FUNCTION_BLOCK EL3151
VAR
	_io : EL3xx1_Data;
	{attribute addProperty Name "WcState"}
	_wcState : WcStateInputToggle;
	{attribute addProperty Name "Info data"}
	_infoData : InfoDataAds;
END_VAR

PROPERTY IO : REFERENCE TO EL3xx1_Data
GET
IO REF= _io;
END_GET
END_PROPERTY

PROPERTY WcState : REFERENCE TO WcStateInputToggle
GET
WcState REF= _wcState;
END_GET
END_PROPERTY

END_FUNCTION_BLOCK

(* stored: Version 1.1.0.1, ProductVersion 3.1.4024.9
   POU EL3151: Id {22b502fe-7958-0569-1483-5dafe6f15503}, SpecialFunc None
   Property IO: Id {252b1368-1d3e-0cca-3519-08f623888de6}
   Get Get: Id {f1316b19-ce5a-0a21-0a14-c32ff0a7ba02}
   Property WcState: Id {1996d15e-1d9a-0410-2aba-a42924e414d7}
   Get Get: Id {d269cb3f-0924-000b-2601-e76b2abb511f} *)
